FUNCTION_BLOCK BUTTON_HMI (* Service Interface Function Block Type *)
  (* Standard: 61499-2 *)
  (* Version 0.0, 19/11/2012, vvya002, nxtControl GmbH, template *)
  PACKAGE Main;
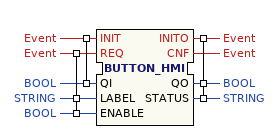
  EVENT_INPUT
    INIT WITH QI;
    REQ WITH LABEL, ENABLE;
  END_EVENT
  EVENT_OUTPUT
    INITO WITH QO, STATUS;
    CNF;
  END_EVENT
  VAR_INPUT
    QI : BOOL;
    LABEL : STRING;
    ENABLE : BOOL;
  END_VAR
  VAR_OUTPUT
    QO : BOOL; (* Event Output Qualifier *)
    STATUS : STRING; (* Service Status *)
  END_VAR
END_FUNCTION_BLOCK
